{attribute 'reflection'}
FUNCTION_BLOCK T_Notification IMPLEMENTS I_Notification
VAR
    {attribute 'instance-path'} {attribute 'no_init'}
    FullName : T_MaxString; // Automatically initialised with the full name of the instance   
    
    EventHandlers : T_ListONotificationHandlers(Capacity := 5);
    
    _Name : T_MaxString; // stripped version
    _Args : T_Stream(StreamLength := 8);
    _NotificationId : UDINT := 999999; // initialise with unlikely notification id to catch cases where it is not initialised by client code
END_VAR

METHOD AddNotificationHandler : I_Notification
VAR_INPUT
    Handler : I_NotificationHandler;
END_VAR
EventHandlers.AddHandler(Handler);
AddNotificationHandler := THIS^;
END_METHOD

PROPERTY PUBLIC Args : I_StreamWriter
GET
Args := _Args;
END_GET
END_PROPERTY

METHOD ClearNotificationHandlers : I_Notification
EventHandlers.Clear();
ClearNotificationHandlers := THIS^;
END_METHOD

METHOD FB_init : BOOL
VAR_INPUT
	bInitRetains : BOOL; // if TRUE, the retain variables are initialized (warm start / cold start)
	bInCopyCode : BOOL;  // if TRUE, the instance afterwards gets moved into the copy code (online change)
END_VAR
VAR
    
END_VAR
THIS^._Name := stripName(FullName);
END_METHOD

PROPERTY Name : T_MaxString
GET
Name := _Name;
END_GET
END_PROPERTY

PROPERTY NotificationId : UDINT
GET
NotificationId := _NotificationId;
END_GET
SET
_NotificationId := NotificationId;
END_SET
END_PROPERTY

METHOD Raise
VAR
    Handler : I_NotificationHandler;
    i : UDINT;
END_VAR
IF EventHandlers.Count > 0 THEN
    FOR i := 0 TO EventHandlers.Count - 1 DO
        Handler := EventHandlers.GetHandler(i);
        IF Handler <> 0 THEN
            _Args.Seek(0); // to ensure that each handler reads args from start of the stream
            Handler.OnNotificationReceived(
                NotificationId   := _NotificationId,
                NotificationName := _Name,
                Args             := _Args);
        END_IF
    END_FOR
END_IF
_Args.Clear(); // to leave event args empty for next time event is raised
END_METHOD

METHOD SetNotificationId : I_Notification
VAR_INPUT
    NotificationId : UDINT;
END_VAR
_NotificationId   := NotificationId;
SetNotificationId := THIS^;
END_METHOD

METHOD PRIVATE stripName : T_MaxString
VAR_INPUT
    FullName : T_MaxString;
END_VAR
VAR
    StringSplitter : T_StringSplitter;
    Result : T_MaxString;
END_VAR
StringSplitter.Init(
    Str := FullName,
    Delim1 := '.',
    Delim2 := '');
    
WHILE StringSplitter.HasMore() DO
    Result := StringSplitter.GetNext(); // to get last sub-section
END_WHILE

StripName := Result;
END_METHOD

END_FUNCTION_BLOCK

(* stored: Version 1.1.0.1, ProductVersion 3.1.4024.4
   POU T_Notification: Id {34c3e11c-b24b-47fd-988a-f99b18a3f2ec}, SpecialFunc None
   Folder Methods: Id {b30ccf79-62ad-46da-a613-c3db6aa14265}
   Folder Properties: Id {376ef0d4-0330-4112-ac16-061d4f2c6035}
   Method AddNotificationHandler: Id {bad47bb4-23ca-4961-a375-b50fdcef3f1a}
   Property Args: Id {81d2c015-f4cb-4582-8ade-a9757b20d5f0}
   Get Get: Id {74639c3f-ebbc-4092-a1f0-5bf037d256a8}
   Method ClearNotificationHandlers: Id {505e6c2b-db1c-4664-9c9e-5c68fcd6cf2b}
   Method FB_init: Id {55e8da39-7c08-4ae7-9330-aaaffad30746}
   Property Name: Id {27a7f7fd-434e-44a7-a257-8a5e63757ddb}
   Get Get: Id {2250062e-718a-417d-ae7e-c7de3531fddb}
   Property NotificationId: Id {f5eb17d4-f0fb-461e-9e8c-6b23479d198c}
   Get Get: Id {7bf505f5-71a4-4cb1-846e-61f59c84ca73}
   Set Set: Id {179ca6ef-e429-497b-92fc-87fee1e765cd}
   Method Raise: Id {96b98869-baef-4dec-8667-b534757ed3a1}
   Method SetNotificationId: Id {d766547e-9576-4401-9528-294aa94bb483}
   Method stripName: Id {44142b3a-8330-47f9-8fd3-23d977d60ed1} *)
